VISUALIZATION VISU_State_gray_green  // 12x17
VAR_IN_OUT
	state : BOOL;
END_VAR
    Ellipse (0,5 10x10), colour toggle: state
END_VISUALIZATION

(* stored: Version 1.1.0.1, ProductVersion 3.1.0.36
   Visu VISU_State_gray_green: Id {d20d0e7f-7f4e-458d-9ec7-f50633309079} *)
